Fanuc TP program (LS listing): OPEN_T1.LS

/PROG  OPEN_T1	  Macro
/ATTR
OWNER		= MNEDITOR;
COMMENT		= "";
PROG_SIZE	= 162;
CREATE		= DATE 25-07-07  TIME 18:38:56;
MODIFIED	= DATE 25-07-07  TIME 19:12:18;
FILE_NAME	= ;
VERSION		= 0;
LINE_COUNT	= 2;
MEMORY_SIZE	= 526;
PROTECT		= READ_WRITE;
TCD:  STACK_SIZE	= 0,
      TASK_PRIORITY	= 50,
      TIME_SLICE	= 0,
      BUSY_LAMP_OFF	= 0,
      ABORT_REQUEST	= 0,
      PAUSE_REQUEST	= 0;
DEFAULT_GROUP	= *,*,*,*,*;
CONTROL_CODE	= 00000000 00000000;
/MN
   1:  RO[3:ON :open T1]=ON ;
   2:  //RO[4:OFF:close T1]=OFF ;
/POS
/END
